// TIA Portal project "Karşılaştırıcılar Uygulama" (V17)

(* hardware
DEVICE "S71500/ET200MP-Station_1"  S7-1500 station
   slot 0: "Profilschiene_0"  6ES7 590-1***0-0AA0
   slot 1: "PLC_1"  CPU 1511-1 PN  6ES7 511-1AK00-0AB0  V1.8
   slot 2: "AI 8xU/I/RTD/TC ST_1"  AI 8xU/I/RTD/TC ST  6ES7 531-7KF00-0AB0  V2.0
   slot 3: "AI 8xU/I/RTD/TC ST_2"  AI 8xU/I/RTD/TC ST  6ES7 531-7KF00-0AB0  V2.0
   slot 4: "AI 8xU/I/RTD/TC ST_3"  AI 8xU/I/RTD/TC ST  6ES7 531-7KF00-0AB0  V2.0
   slot 5: "AI 8xU/I/RTD/TC ST_4"  AI 8xU/I/RTD/TC ST  6ES7 531-7KF00-0AB0  V2.0
   slot 6: "DI 16x24VDC BA_1"  DI 16x24VDC BA  6ES7 521-1BH10-0AA0  V1.0
*)

// ===== PLC "PLC_1"  CPU 1511-1 PN =====

VAR_GLOBAL   // PLC tag table "Standard-Variablentabelle"
   "ŞALTER" AT %E0.0 : Bool;
   "1.KONVEYOR" AT %A0.0 : Bool;
   "START" AT %E0.1 : Bool;
   "Tag_1" AT %M0.0 : Bool;
   "STOP" AT %I0.2 : Bool;
   "Tag_3" AT %M10.0 : Bool;
   "Tag_4" AT %ID30 : DWord;
   "Tag_5" AT %M0.1 : Bool;
   "2.KONVEYOR" AT %Q0.1 : Bool;
   "Tag_6" AT %Q0.3 : Bool;
   "İTİCİ BANT" AT %Q0.2 : Bool;
   "SENSOR" AT %I0.3 : Bool;
   "Tag_9" AT %M1.3 : Bool;
END_VAR

// folder: System blocks/Program resources

DATA_BLOCK "IEC_Timer_0_DB"   // DB1
{ S7_Optimized_Access := 'TRUE' }
AUTHOR : Simatic
FAMILY : IEC
NAME : IEC_TMR
VERSION : 1.0
// stored: InstanceOfName IEC_TIMER
"IEC_TIMER"
BEGIN
END_DATA_BLOCK

// folder: (top level)

FUNCTION "MHJ-PLC-Lab-Function-S71500" : Void   // FC9000, SCL
{ S7_Optimized_Access := 'TRUE' }
VERSION : 0.1
   VAR_TEMP
      Value : Byte;
      ForCounter : Int;
   END_VAR
   VAR CONSTANT
      Value_01_DW : DWord := 16#1223_5486;
      Value_02_DW : DWord := 16#A6C9_D1F5;
   END_VAR
BEGIN

   #Value:=PEEK(area := 16#82,
        dbNumber := 0,
        byteOffset := 511);
   #Value := #Value + 1;

   POKE(area := 16#82,
        dbNumber := 0,
        byteOffset := 511,
        value := #Value);

   POKE(area := 16#82,
        dbNumber := 0,
        byteOffset := 1016,
        value := #Value_01_DW);
   POKE(area := 16#82,
        dbNumber := 0,
        byteOffset := 1020,
        value := #Value_02_DW);

   FOR #ForCounter := 0 TO 63 DO
       #Value:=PEEK(area := 16#1,
            dbNumber := 0,
            byteOffset := #ForCounter);
       POKE(area := 16#81,
            dbNumber := 0,
            byteOffset := #ForCounter,
            value := #Value);
   END_FOR;
   #Value := PEEK(area := 16#1,
                  dbNumber := 0,
                  byteOffset := 512);
   POKE(area := 16#82,
        dbNumber := 0,
        byteOffset := 512,
        value := #Value);
END_FUNCTION

ORGANIZATION_BLOCK "Main"   // OB1, LAD, ProgramCycle
TITLE = "Main Program Sweep (Cycle)"
{ S7_Optimized_Access := 'TRUE' }
VERSION : 0.1
   VAR_INPUT
      Initial_Call : Bool;   // Initial call of this OB
      Remanence : Bool;   // =True, if remanent data are available
   END_VAR
   VAR_TEMP   // added for the SCL form of the ladder/FBD networks
      _w1 : Bool;
      _w2 : Bool;
   END_VAR
BEGIN

REGION Network 1
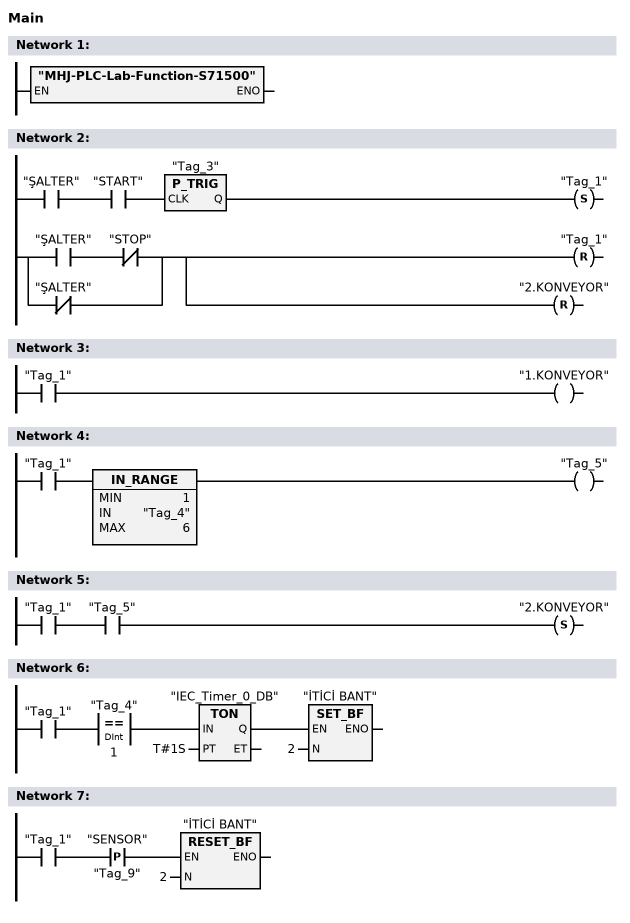
   RUNG wire#powerrail
      "MHJ-PLC-Lab-Function-S71500"()
   END_RUNG
   // the same network as SCL:
   "MHJ-PLC-Lab-Function-S71500"();
END_REGION

REGION Network 2
   RUNG wire#powerrail
      Contact( "ŞALTER" )
      Contact( "START" )
      P_Trig( "Tag_3" )
      S_Coil( "Tag_1" )
   END_RUNG
   RUNG wire#powerrail
      Contact( "ŞALTER" )
      I_Contact( "STOP" )
      wire#w1
      R_Coil( "Tag_1" )
   END_RUNG
   RUNG wire#powerrail
      I_Contact( "ŞALTER" )
   END_RUNG wire#w1
   RUNG wire#w1
      R_Coil( "2.KONVEYOR" )
   END_RUNG
   // the same network as SCL:
   #_w1 := "ŞALTER" AND "START";
   #_w2 := #_w1 AND NOT "Tag_3";   // rising edge
   "Tag_3" := #_w1;
   IF #_w2 THEN "Tag_1" := TRUE; END_IF;
   IF ("ŞALTER" AND NOT "STOP") OR NOT "ŞALTER" THEN
       "Tag_1" := FALSE;
       "2.KONVEYOR" := FALSE;
   END_IF;
END_REGION

REGION Network 3
   RUNG wire#powerrail
      Contact( "Tag_1" )
      Coil( "1.KONVEYOR" )
   END_RUNG
   // the same network as SCL:
   "1.KONVEYOR" := "Tag_1";
END_REGION

REGION Network 4
   RUNG wire#powerrail
      Contact( "Tag_1" )
      { S7_Templates := "SrcType := DInt" } InRange(min := 1, in := "Tag_4", max := 6)
      Coil( "Tag_5" )
   END_RUNG
   // the same network as SCL:
   "Tag_5" := "Tag_1" AND (1 <= "Tag_4") AND ("Tag_4" <= 6);
END_REGION

REGION Network 5
   RUNG wire#powerrail
      Contact( "Tag_1" )
      Contact( "Tag_5" )
      S_Coil( "2.KONVEYOR" )
   END_RUNG
   // the same network as SCL:
   IF "Tag_1" AND "Tag_5" THEN "2.KONVEYOR" := TRUE; END_IF;
END_REGION

REGION Network 6
   // no SCL statement known for SBitfield: written as a call
   "IEC_Timer_0_DB".TON(IN := "Tag_1" AND ("Tag_4" = 1), PT := T#1S);
   IF "IEC_Timer_0_DB".Q THEN SET_BF(operand := "İTİCİ BANT", n := 2); END_IF;
END_REGION

REGION Network 7
   // no SCL statement known for RBitfield: written as a call
   #_w1 := "Tag_1" AND "SENSOR" AND NOT "Tag_9";   // rising edge of "SENSOR"
   "Tag_9" := "SENSOR";
   IF #_w1 THEN RESET_BF(operand := "İTİCİ BANT", n := 2); END_IF;
END_REGION
END_ORGANIZATION_BLOCK